(* CODESYS project Observer_Application.project

Project tree, tasks and I/O mapping:
  Device : CODESYS Control for Raspberry Pi SL, 3S - Smart Software Solutions GmbH, version 3.5.9.40
    application Application
      libraries: Standard, * (System)
      task MainTask (cyclic, interval t#10ms, priority 1) calls PLC_PRG
      task VISU_TASK (cyclic, interval 100 ms, priority 31) calls VisuElems.Visu_Prg
      program PLC_PRG [ST]
      interface Observer_Interface: update
      interface Subject_Interface: registerObserver, removeObserver, notifyObservers
      function block ConcreteSubject [ST]: registerObserver, removeObserver, notifyObservers, Set_observedINT
      function block ConcreteObserver [ST]: update, fb_init
      global variables Observer_Config
      visualisation Visualization
    SoftMotion General Axis Pool
    GPIOs_A_B : GPIOs A/B, 3S - Smart Software Solutions GmbH, version 1.1.1.10
        unmapped channels: digital inputs (GPIO0..GPIO31), digital outputs (GPIO0..GPIO31)
    I²C
    SPI
    Onewire
    Camera device
      <Empty>
  libraries: VisuSymbols, 3.5.10.0 (System)
  text list GlobalTextList
*)

// Device/Application/Observer_Config
{attribute 'qualified_only'}
VAR_GLOBAL CONSTANT
	//Constant variable to determine the size of the observerList array.
	//This variable is the MAXIMUM number of observer objects that can be subscribed to the subject
	C_MAX_OBSERVER_NUM : INT := 10;
	//Pointer to a null Observer_Interface object.
	//This pointer is used to validate the addresses to be used. These addresses must to be <> than this null pointer to have effect in the code
	nullPointerToObserver : Observer_Interface;
END_VAR

// Device/Application/PLC_PRG
//Main program
PROGRAM PLC_PRG
VAR
	//Subject instance declaration
	realSubject 	: ConcreteSubject;
	
	//Observer instance declaration
	realObserver 	: ConcreteObserver;
	
	//Observer instance declaration
	realObserver2 	: ConcreteObserver;
	
	//Observer instance declaration
	realObserver3 	: ConcreteObserver;

END_VAR

//THE PLC_PRG handles the instanciation of the Subject and Observers in order to be used by the Visualization element

//The Visualization element can handle the registration and deregistration of observers.
//The Visualization element is also in charge of the realSubject.intToBeObserved value changes.
//By default, no observes is registered, so if there is a change on the subject's state, no observer will receive the notification unless they are registered by the client (Visualization element).

END_PROGRAM

// Device/Application/ConcreteSubject
{attribute 'enable_dynamic_creation'}
//Subject class

FUNCTION_BLOCK ConcreteSubject IMPLEMENTS Subject_Interface
VAR_INPUT
END_VAR
VAR_OUTPUT
END_VAR
VAR CONSTANT
	//Constant value to identify the maximum number of observers in the observerList array
	maxObservers :INT := Observer_Config.C_MAX_OBSERVER_NUM;
END_VAR
VAR
	
//Array of observers suscribed to the subject. 
	observerList : ARRAY[1..maxObservers] OF Observer_Interface;
	
//Field to be watch by the observers
	intToBeObserved : INT;
END_VAR

//Method to register observers
METHOD registerObserver
VAR_INPUT
//Observer to be registered
	newObserver : Observer_Interface;
END_VAR
VAR
	//Local value to circle the observerList array
	index : INT :=0;
	bObserverRegistered : BOOL := FALSE;
	bFirstFreeSlot : BOOL := FALSE;
	firstFreeSlot : INT := 0;
END_VAR
//Verifies if the passed observer has a valid address <> null
IF newObserver <> Observer_Config.nullPointerToObserver
	THEN
	//If so, then starting in the index 1 until the maximum number of observers DO
	FOR index :=1 TO THIS^.maxObservers BY 1 DO
		//Verify if the Observer to be registered is already registered
		IF THIS^.observerList[index] = newObserver
			THEN
			//If so, the a message will be sent to the client and a break out of the FOR loop is made
			bObserverRegistered := TRUE;
			index := THIS^.maxObservers;
			//If the Observer is not already registered in this index, then we verify if a free slot has not been found yet
			//If a free slot has been found, it will just ignore this statement
			ELSIF bFirstFreeSlot = FALSE
				THEN
				//If a free slot has not been found, we verify if the current index is an empty slot in the observerList array
				IF	THIS^.observerList[index] = Observer_Config.nullPointerToObserver
					THEN	
					//If the current address is indeed a free slot inside the observerList array, then we have found the first free slot inside the array
					//The boolean flag of FreeSlotFound is set to TRUE and we save the current index, this being the index of the first free slot inside the array				
					bFirstFreeSlot := TRUE;
					firstFreeSlot := index;
				END_IF	
		END_IF
	END_FOR
	
	//Once the FOR loop has ended, we have all the information to register or not the passed observer.
	
	//If the observer is already registered, we send a message to the client 
	IF bObserverRegistered
		THEN
		(*Send an arror to the Client "The Observer is already registered to the Subject" *)
		
	// Once we know the observer has not been registered, we verify the existance of an empty slot in the observerList array
	ELSIF bFirstFreeSlot
		THEN
		//Once the empty slot is found, saves the observer object to the array of observers suscribed to the subject in the firstFreeSlot previously found
		THIS^.observerList[firstFreeSlot] := newObserver;
		//Now, the new observer is notified ob the status of the intToBeObserved
		THIS^.observerList[firstFreeSlot].update(THIS^.intToBeObserved);
	
	ELSE
		//This statement will only be triggered if the passed observer has not been registered and it was impossible to find a free slot in the observerList array
		//Then we send a message to the client
		
		(* PRINT ERROR LOG "NO OBSERVER SLOT AVAILABLE" *)
	END_IF
END_IF
END_METHOD

//Method to unsuscribe observers
METHOD removeObserver
VAR_INPUT
//Observer to be romeved
	deleteObserver : Observer_Interface;
END_VAR
VAR
	//Local value to circle the observerList array
	index : INT := 0;
END_VAR
//Verifies if the passed observer has a valid address <> null
IF deleteObserver <> Observer_Config.nullPointerToObserver
	THEN
	//If so, then starting in the index 1 until the maximum number of observers DO
	FOR index := 1 TO THIS^.maxObservers BY 1 DO
		//Verify if theobserver to be removed is in the current index
		IF THIS^.observerList[index] = deleteObserver
			THEN
			//If so, then overridethe current index with a nullPointer
			THIS^.observerList[index] := Observer_Config.nullPointerToObserver;	
			//If for some reason the observer is registered in two or more array slots, the FOR loop will override every slot until the maximum number of observers is reached.
			//This could be avoided by ensuring there can not be two slots with the same address with the registerObserver method
			// if there cannot be two or more slots with the same address inside the array, then we can force a break out of the For loop, otherwise we have to comment the next line to finish the For loop and check the whole observerList array.
			index := THIS^.maxObservers;
		END_IF
	END_FOR
END_IF
END_METHOD

//Method to send the updates to the observers
METHOD notifyObservers
VAR	
//Local value to ensure every observer got the update method
	index: INT := 0;
END_VAR
//For loop to use the update method of every observer suscribed to the subject
//Starring with the index 1 of the array until the total amount of observers DO:
FOR index := 1 TO THIS^.maxObservers BY 1 DO
	//Verify the current address in the array is a valid address
	IF THIS^.observerList[index] <> Observer_Config.nullPointerToObserver
		THEN
		//If so, then use the object stored in the array of observer suscribed (Observer objects)
		// and call its own update method passing the change on the observed field
		THIS^.observerList[index].update(THIS^.intToBeObserved);
	END_IF
END_FOR
END_METHOD

//Simple SET method to modify and send updates to the observers

METHOD Set_observedINT
VAR_INPUT
	
	//Passed number to be written on the observed field
	num : INT;
END_VAR
//Set the correct value to the observed field
THIS^.intToBeObserved := num;

//Call the notify method of the subject to send the updates to the observers suscribed
THIS^.notifyObservers();
END_METHOD

END_FUNCTION_BLOCK

// Device/Application/Subject_Interface
//Interface to be implemented by every subject class

INTERFACE Subject_Interface

//Method to register a new observer

METHOD registerObserver
VAR_INPUT
	
//Observer to be registered to the subject
	newObserver : Observer_Interface;
END_VAR
END_METHOD

//Method to remove observers

METHOD removeObserver
VAR_INPUT
	
//Observer to be unsuscribed to the subject
	deleteObserver : Observer_Interface;
END_VAR
END_METHOD

//Method to notify the observers of changes on the Subject

METHOD notifyObservers
VAR_INPUT
END_VAR
END_METHOD

END_INTERFACE

// Device/Application/Observer_Interface
//Interface to be implemented by every observer class

INTERFACE Observer_Interface

//Method to update the values from the subject

METHOD update

VAR_INPUT
	
	//Variable to be passed from the subject intToBeObserved
	num : INT;
END_VAR
END_METHOD

END_INTERFACE

// Device/Application/ConcreteObserver
{attribute 'enable_dynamic_creation'}

//Observer class
FUNCTION_BLOCK ConcreteObserver IMPLEMENTS Observer_Interface
VAR_INPUT
END_VAR
VAR_OUTPUT
END_VAR
VAR
	
//Field to recive updates from the subject
	intObserved : INT;

//Not really needed, just keeps the order of which observer called the constructor first
	observerID : INT;
END_VAR
VAR_STAT
	
//Not really needed, just keeps the record of how many times the constructor was called
	observerIDTracker : INT;
END_VAR

//Method called to get the updates from the subject

METHOD update
VAR_INPUT
	
//Value to be passed from the subject
	num : INT;
END_VAR
//Sets the specific field for the observed value
THIS^.intObserved := num;
END_METHOD

METHOD fb_init
VAR_INPUT
	bInitRetains : BOOL; // TRUE: the Retain-variables are initialized (reset warm / reset cold)
	bInCopyCode : BOOL;  // TRUE  the instance will be copied to the copy-code afterward (online change)	
END_VAR
//Constructor of the observer class
//It is not really needed the constructor here doesn't affect the function of the observer pattern

//Increments the number of observers that have used the constructor
THIS^.observerIDTracker := THIS^.observerIDTracker + 1;

//Sets the unique observerID according to the number of observers
THIS^.observerID := THIS^.observerIDTracker;
END_METHOD

END_FUNCTION_BLOCK

// Device/Application/Visualization
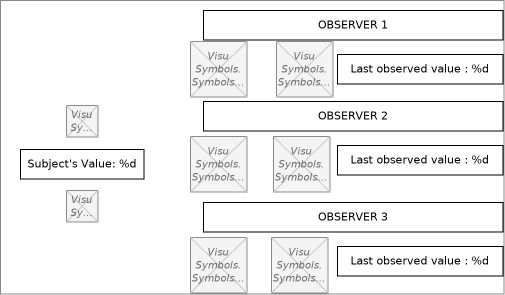
VISUALIZATION Visualization  // 505x295
//THE PLC_PRG handles the instanciation of the Subject and Observers in order to be used by the Visualization element
//The Visualization element can handle the registration and deregistration of observers.
//The Visualization element is also in charge of the realSubject.intToBeObserved value changes.
//By default, no observes is registered, so if there is a change on the subject's state, no observer will receive the notification unless they are registered by the client (Visualization element).
    Image (66,190 32x32), image: VisuSymbols.Symbols.ArrowBoldDown
        OnMouseDown: execute { PLC_PRG.realSubject.Set_observedINT(PLC_PRG.realSubject.intToBeObserved - 1); }
    Image (66,105 32x32), image: VisuSymbols.Symbols.ArrowBoldUp
        OnMouseDown: execute { PLC_PRG.realSubject.Set_observedINT(PLC_PRG.realSubject.intToBeObserved + 1); }
    RoundedRectangle (20,149 124x30), "Subject's Value: %d", text variable: PLC_PRG.realSubject.intToBeObserved
    Image (190,41 57x56), tooltip "follow subject", image: VisuSymbols.Symbols.AddUser
        OnMouseDown: execute { PLC_PRG.realSubject.registerObserver(PLC_PRG.realObserver); }
    Image (276,41 57x56), tooltip "unfollow subject", image: VisuSymbols.Symbols.DeleteUser
        OnMouseDown: execute { PLC_PRG.realSubject.removeObserver(PLC_PRG.realObserver); }
    RoundedRectangle (203,10 300x30), "OBSERVER 1"
    RoundedRectangle (337,54 166x30), "Last observed value : %d", text variable: PLC_PRG.realObserver.intObserved
    Image (190,136 57x56), tooltip "follow subject", image: VisuSymbols.Symbols.AddUser
        OnMouseDown: execute { PLC_PRG.realSubject.registerObserver(PLC_PRG.realObserver2); }
    Image (273,136 57x56), tooltip "unfollow subject", image: VisuSymbols.Symbols.DeleteUser
        OnMouseDown: execute { PLC_PRG.realSubject.removeObserver(PLC_PRG.realObserver2); }
    RoundedRectangle (203,101 300x30), "OBSERVER 2"
    RoundedRectangle (337,145 166x30), "Last observed value : %d", text variable: PLC_PRG.realObserver2.intObserved
    Image (190,237 57x56), tooltip "follow subject", image: VisuSymbols.Symbols.AddUser
        OnMouseDown: execute { PLC_PRG.realSubject.registerObserver(PLC_PRG.realObserver3); }
    Image (271,237 57x56), tooltip "unfollow subject", image: VisuSymbols.Symbols.DeleteUser
        OnMouseDown: execute { PLC_PRG.realSubject.removeObserver(PLC_PRG.realObserver3); }
    RoundedRectangle (203,202 300x30), "OBSERVER 3"
    RoundedRectangle (337,246 166x30), "Last observed value : %d", text variable: PLC_PRG.realObserver3.intObserved
END_VISUALIZATION
